FUNCTION_BLOCK FB_ElementTest EXTENDS TcUnit.FB_TestSuite
VAR
END_VAR


T01_TestCreateAndLinkData ();

METHOD PRIVATE T01_TestCreateAndLinkData
VAR_INPUT
END_VAR

VAR
	bWynik: BOOL;
END_VAR
IF (TcUnit.TEST_ORDERED ('T01_TestCreateAndLinkData')) THEN
	bWynik := GVL_Variable.fbComponent_1.LinkData (stCommonData := gvl.stCommonData);
	AssertTrue (Condition := bWynik, Message := 'T01 - test linkowania zmiennych ');
	GVL_VariableHMI.fbComponentHMI_1.LinkData (stCommonData := GVL.stCommonData);
	AssertTrue (Condition := bWynik, Message := 'T02 - test linkowania zmiennych ');
	
	bWynik := GVL_Variable.fbControlElement_1.LinkData (stCommonData := gvl.stCommonData);
	AssertTrue (Condition := bWynik, Message := 'T03 - test linkowania zmiennych ');
	GVL_VariableHMI.fbControlrElementHMI_1.LinkData (stCommonData := GVL.stCommonData);
	AssertTrue (Condition := bWynik, Message := 'T04 - test linkowania zmiennych ');
	
	bWynik := GVL_Variable.fbGroupElement_1.LinkData (stCommonData := gvl.stCommonData);
	AssertTrue (Condition := bWynik, Message := 'T05 - test linkowania zmiennych ');
	GVL_VariableHMI.fbGroupElementHMI_1.LinkData (stCommonData := GVL.stCommonData);
	AssertTrue (Condition := bWynik, Message := 'T06 - test linkowania zmiennych ');
	
	bWynik := GVL_Variable.fbTopElement_1.LinkData (stCommonData := gvl.stCommonData);
	AssertTrue (Condition := bWynik, Message := 'T07 - test linkowania zmiennych ');
	GVL_VariableHMI.fbTopElementHMI_1.LinkData (stCommonData := GVL.stCommonData);
	AssertTrue (Condition := bWynik, Message := 'T08 - test linkowania zmiennych ');
	
(*	Test czy itf są przepisane	*)	

	AssertTrue (Condition := GVL_VariableHMI.fbComponentHMI_1.GetIsInit (), Message := 'T09 - Blad inicjalizacji');
	AssertTrue (Condition := GVL_VariableHMI.fbControlrElementHMI_1.GetIsInit (), Message := 'T10 - Blad inicjalizacji');
	AssertTrue (Condition := GVL_VariableHMI.fbGroupElementHMI_1.GetIsInit (), Message := 'T11 - Blad inicjalizacji');
	AssertTrue (Condition := GVL_VariableHMI.fbTopElementHMI_1.GetIsInit (), Message := 'T12 - Blad inicjalizacji');
	
		
	TcUnit.TEST_FINISHED ();
END_IF
END_METHOD

END_FUNCTION_BLOCK

(* stored: Version 1.1.0.1, ProductVersion 3.1.4024.15
   POU FB_ElementTest: Id {3cbac2ab-f33e-495d-b5c8-b7ba1b9f5011}, SpecialFunc None
   Method T01_TestCreateAndLinkData: Id {d3c385be-3c77-42c2-89b9-e1b9a0939a42} *)
